DATA_BLOCK "DB_Global"
{ S7_Optimized_Access := 'FALSE' }
VERSION : 0.1
NON_RETAIN
// 2. GLOBAL DATA (Pure Data only)
   STRUCT
      Sys { ExternalAccessible := 'False'; ExternalVisible := 'False'; ExternalWritable := 'False'; S7_SetPoint := 'False'} : "UDT_Sys_Info";
      c_stDI_Mode { ExternalAccessible := 'False'; ExternalVisible := 'False'; ExternalWritable := 'False'} : Struct
         None { ExternalAccessible := 'False'; ExternalVisible := 'False'; ExternalWritable := 'False'} : Int;
         NOpen { ExternalAccessible := 'False'; ExternalVisible := 'False'; ExternalWritable := 'False'} : Int;
         NClose { ExternalAccessible := 'False'; ExternalVisible := 'False'; ExternalWritable := 'False'} : Int;
         Disabled { ExternalAccessible := 'False'; ExternalVisible := 'False'; ExternalWritable := 'False'} : Int;
      END_STRUCT;
   END_STRUCT;


BEGIN
   Sys.CycleTime_ms_INT := 10;
   Sys.CycleTime_ms_REAL := 10.0;
   c_stDI_Mode.NOpen := 1;
   c_stDI_Mode.NClose := 2;
   c_stDI_Mode.Disabled := 3;

END_DATA_BLOCK

